// SIMATIC S7-200 project (STEP 7-Micro/WIN), CPU 224XP REL 02.01

SYMBOL_TABLE 输入
一号泵故障            I0.0     // 1号水泵工频故障
二号泵故障            I0.1     // 2号水泵工频故障
三号泵故障            I0.2     // 3号水泵工频故障
一号泵变频运行反馈        I0.3     // 1号水泵变频接触器辅助常开触点
一号泵工频运行反馈        I0.4     // 1号水泵工频接触器辅助常开触点
二号泵变频运行反馈        I0.5     // 2号水泵变频接触器辅助常开触点
二号泵工频运行反馈        I0.6     // 2号水泵工频接触器辅助常开触点
三号泵变频运行反馈        I0.7     // 3号水泵变频接触器辅助常开触点
三号泵工频运行反馈        I1.0     // 3号水泵工频接触器辅助常开触点
变频运行             I1.1     // 变频器准备就绪
变频故障             I1.2     // 变频器故障
自动切换             I1.3     // 变频器达到最大频率
急停               I1.5     // 急停
远方起动             I2.0     // 远方起动系统
水位下限             I2.1     // 水源低水位限位开关
水位上限             I2.2     // 水源高水位限位开关
供水方式             I2.3     // 生活用水/消防用水切换，触点常开为生活用水工作方式
压力测量             AIW0     // 管网压力传感器测量值:4-20mA
END_SYMBOL_TABLE

SYMBOL_TABLE 输出
一号泵变频运行          Q0.0     // 1号水泵变频接触器
一号泵工频运行          Q0.1     // 1号水泵工频接触器
二号泵变频运行          Q0.2     // 2号水泵变频接触器
二号泵工频运行          Q0.3     // 2号水泵工频接触器
三号泵变频运行          Q0.4     // 3号水泵变频接触器
三号泵工频运行          Q0.5     // 3号水泵工频接触器
准备就绪             Q0.6     // 系统准备就绪
报警信号             Q0.7     // 系统报警信号
故障跳闸             Q1.0     // 系统故障跳闸
起动停止             Q1.1     // 变频器起动/停止
供水电磁阀            Q2.0     // 生活用水/消防用水电磁阀控制
频率复位             Q2.1     // 变频器频率复位控制
模拟输出             AQW0     // 变频器模拟输入，PID运算结果: 4-20mA
END_SYMBOL_TABLE

SYMBOL_TABLE PLC內部继电器
允许启动             M1.0     // 系统准备就绪指示
低水位报警            M1.1     // 低水位报警铃声，信号指示
变频报警             M1.2     // 变频器报警铃声，信号指示
火灾报警             M1.3     // 火灾报警铃声，信号指示
HMI急停            M1.5     // 触摸屏急停按钮
远方变频起动自保         M1.6     // 远方变频起动信号自保持
故障结束脉冲           M0.0     // 故障结束脉冲信号
变频起动脉冲           M0.1     // 泵变频启动脉冲
水泵轮换             M0.3     // 倒泵变频启动脉冲
复位变频运行脉冲         M0.4     // 复位当前变频泵运行脉冲
当前泵工频            M0.5     // 当前泵工频运行启动脉冲
新增泵变频            M0.6     // 新泵变频启动脉冲
工变频切换1           M2.0     // 水泵工频/变频转换逻辑控制
工变频切换2           M2.1     // 水泵工频/变频转换逻辑控制
工变频切换3           M2.2     // 水泵工频/变频转换逻辑控制
系统故障             M3.0     // 故障汇总
低水位自保            M3.1     // 低水位自保，高水位复位解除
低水位消铃            M3.2     // 低水位报警铃声消音
变频报警消铃           M3.3     // 变频器故障报警铃声消音
火灾报警消铃           M3.4     // 火灾报警铃声消音
一号泵故障指示          M3.5     // 1号水泵电机过载
二号泵故障指示          M3.6     // 2号水泵电机过载
三号泵故障指示          M3.7     // 3号水泵电机过载
故障复位             M4.1     // 故障自锁信号解除
系统报警指示           M4.2     // 报警汇总
报警确认             M4.3     // 报警自锁信号解除
消铃按钮             M4.4     // 报警铃声信号解除
试灯按钮             M4.5     // 检查报警灯光回路
本地/远方            M5.0     // 触摸屏控制/远方集中控制选择: 默认为本地控制
手动/自动            M5.1     // 工频手动/变频自动: 默认为自动控制
一号泵起动按钮          M5.2     // 触摸屏上1号泵起动按钮
一号泵停止按钮          M6.0     // 触摸屏上1号泵停止按钮
一号泵自保持           M6.1     // 1号泵起动信号自保持
二号泵起动按钮          M6.2     // 触摸屏上2号泵起动按钮
二号泵停止按钮          M6.3     // 触摸屏上2号泵停止按钮
二号泵自保持           M6.4     // 2号泵起动信号自保持
三号泵起动按钮          M6.5     // 触摸屏上3号泵起动按钮
三号泵停止按钮          M6.6     // 触摸屏上3号泵停止按钮
三号泵自保持           M6.7     // 3号泵起动信号自保持
                 M7.0     // 触摸屏变频器起动按钮
                 M7.1     // 触摸屏变频器停止按钮
END_SYMBOL_TABLE

SYMBOL_TABLE PLC內部存储器
压力设置             VW0      // 管网压力设置值
水压测量             VW2      // 管网压力传感器测量值
过程变量             VD100
压力给定             VD104
PI计算值            VD108
比例系数             VD112
采样时间             VD116
积分时间             VD120
微分时间             VD124
频率下限             VD204    // 变频运行频率下限值
生活水频率上限          VD208    // 生活供水变频运行频率上限值
消防水频率上限          VD212    // 消防供水变频运行频率上限值
PI调节值            VD250    // PI调节结果存储器
变频泵号             VD300    // 记录当前变频工作泵的泵号
工频泵总数            VD301    // 工频运行泵的总数量
泵轮换时间            VD310    // 变频泵运行时间存储器
工频变频切换1          T33      // 水泵工频/变频转换逻辑时间控制
工频变频切换2          T34      // 水泵工频/变频转换逻辑时间控制
工频变频切换3          T39      // 水泵工频/变频转换逻辑时间控制
工频增泵时间           T37      // 工频泵增泵滤波时间控制
工频减泵时间           T38      // 工频泵减泵滤波时间控制
END_SYMBOL_TABLE

SYMBOL_TABLE S7-200 符号
Always_On        SM0.0    // 始终接通为 ON
First_Scan_On    SM0.1    // 仅第一个扫描周期中接通为 ON
Clock_60s        SM0.4    // 在 1 分钟的循环周期内，接通为 ON 30  秒，关断为 OFF 30 秒
Clock_1s         SM0.5    // 在 1 秒钟的循环周期内，接通为 ON 0.5 秒，关断为 OFF 0.5  秒
Time_0_Intrvl    SMB34    // 定时中断 0 的时间间隔（从 1 至 255，以 1 毫秒为增量）。
END_SYMBOL_TABLE

ORGANIZATION_BLOCK 主程序:OB1
TITLE=程序注释
BEGIN
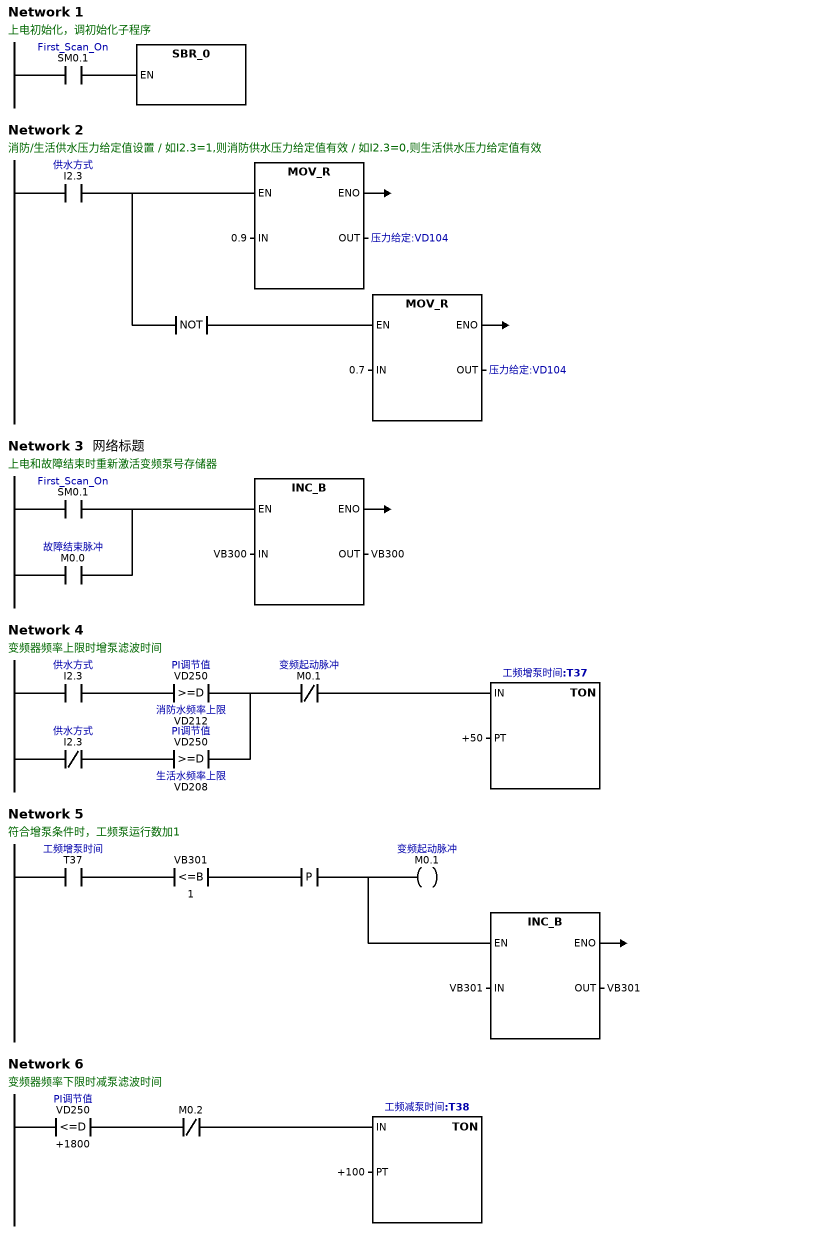
Network 1
// 上电初始化，调初始化子程序
// (network saved uncompiled; LAD cells follow)
// row 0: c0 -| |- First_Scan_On:SM0.1  c1 [SBR_0 EN:=power@row0]
Network 2
// 消防/生活供水压力给定值设置
// 如I2.3=1,则消防供水压力给定值有效
// 如I2.3=0,则生活供水压力给定值有效
// (network saved uncompiled; LAD cells follow)
// row 0: c0 -| |- 供水方式:I2.3 v  c1 --  c2 [MOV_R EN:=power@row0, IN:=0.9, ENO=>power, OUT=>压力给定:VD104]  c3 ->
// row 1: c0 ^v  c2 [box]
// row 2: c0 ^  c1 -|NOT|-  c2 --  c3 [MOV_R EN:=power@row2, IN:=0.7, ENO=>power, OUT=>压力给定:VD104]  c4 ->
// row 3: c3 [box]
Network 3 // 网络标题
// 上电和故障结束时重新激活变频泵号存储器
// (network saved uncompiled; LAD cells follow)
// row 0: c0 -| |- First_Scan_On:SM0.1 v  c1 --  c2 [INC_B EN:=power@row0, IN:=VB300, ENO=>power, OUT=>VB300]  c3 ->
// row 1: c0 -| |- 故障结束脉冲:M0.0 ^  c2 [box]
Network 4
// 变频器频率上限时增泵滤波时间
// (network saved uncompiled; LAD cells follow)
// row 0: c0 -| |- 供水方式:I2.3  c1 -|>=D|- PI调节值:VD250, 消防水频率上限:VD212 v  c2 -|/|- 变频起动脉冲:M0.1  c3 --  c4 [TON 工频增泵时间:T37 IN:=power@row0, PT:=+50]
// row 1: c0 -|/|- 供水方式:I2.3  c1 -|>=D|- PI调节值:VD250, 生活水频率上限:VD208 ^  c4 [box]
Network 5
// 符合增泵条件时，工频泵运行数加1
// (network saved uncompiled; LAD cells follow)
// row 0: c0 -| |- 工频增泵时间:T37  c1 -|<=B|- VB301, 1  c2 -|P|-  v  c3 -( ) 变频起动脉冲:M0.1
// row 1: c2 ^  c3 --  c4 [INC_B EN:=power@row1, IN:=VB301, ENO=>power, OUT=>VB301]  c5 ->
// row 2: c4 [box]
Network 6
// 变频器频率下限时减泵滤波时间
// (network saved uncompiled; LAD cells follow)
// row 0: c0 -|<=D|- PI调节值:VD250, +1800  c1 -|/|- M0.2  c2 --  c3 [TON 工频减泵时间:T38 IN:=power@row0, PT:=+100]
// row 1: c3 [box]
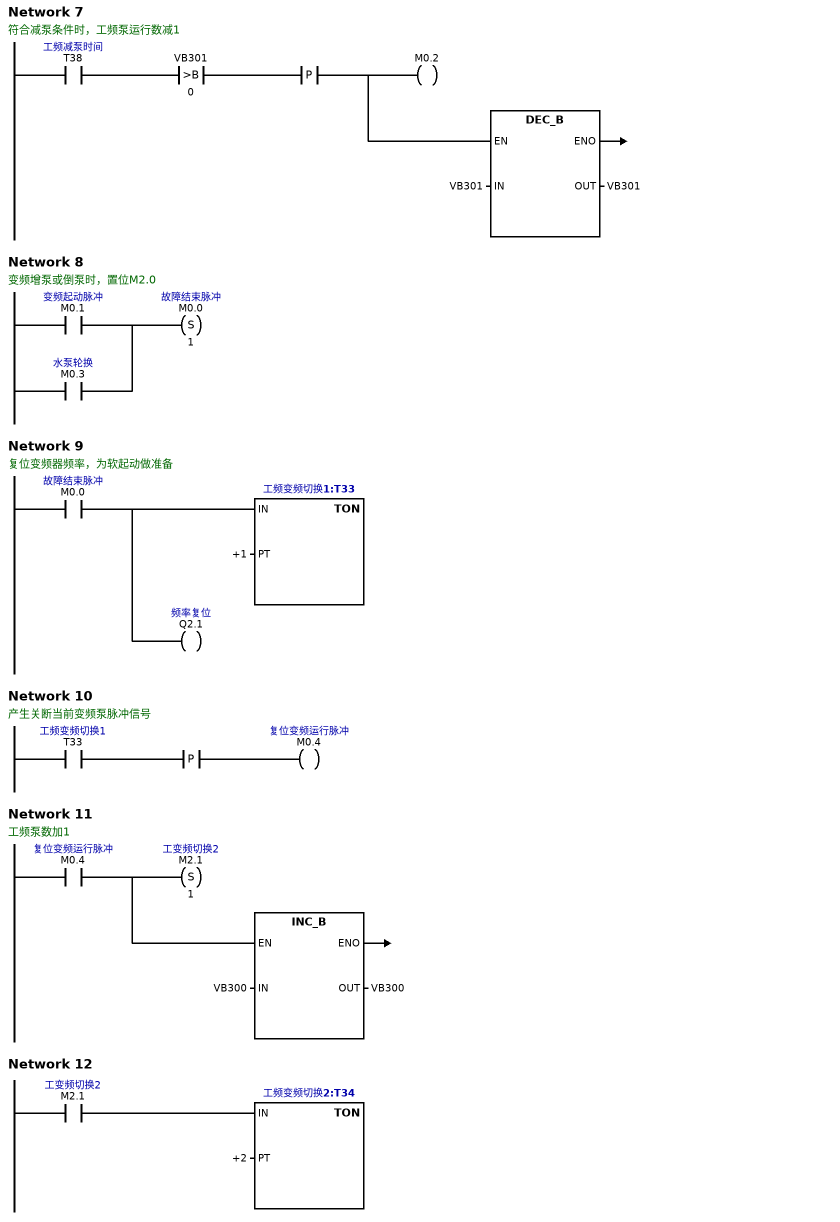
Network 7
// 符合减泵条件时，工频泵运行数减1
// (network saved uncompiled; LAD cells follow)
// row 0: c0 -| |- 工频减泵时间:T38  c1 -|>B|- VB301, 0  c2 -|P|-  v  c3 -( ) M0.2
// row 1: c2 ^  c3 --  c4 [DEC_B EN:=power@row1, IN:=VB301, ENO=>power, OUT=>VB301]  c5 ->
// row 2: c4 [box]
Network 8
// 变频增泵或倒泵时，置位M2.0
// (network saved uncompiled; LAD cells follow)
// row 0: c0 -| |- 变频起动脉冲:M0.1 v  c1 -(S) 故障结束脉冲:M0.0, 1
// row 1: c0 -| |- 水泵轮换:M0.3 ^
Network 9
// 复位变频器频率，为软起动做准备
// (network saved uncompiled; LAD cells follow)
// row 0: c0 -| |- 故障结束脉冲:M0.0 v  c1 --  c2 [TON 工频变频切换1:T33 IN:=power@row0, PT:=+1]
// row 1: c0 ^v  c2 [box]
// row 2: c0 ^  c1 -( ) 频率复位:Q2.1
Network 10
// 产生关断当前变频泵脉冲信号
// (network saved uncompiled; LAD cells follow)
// row 0: c0 -| |- 工频变频切换1:T33  c1 -|P|-  c2 -( ) 复位变频运行脉冲:M0.4
Network 11
// 工频泵数加1
// (network saved uncompiled; LAD cells follow)
// row 0: c0 -| |- 复位变频运行脉冲:M0.4 v  c1 -(S) 工变频切换2:M2.1, 1
// row 1: c0 ^  c1 --  c2 [INC_B EN:=power@row1, IN:=VB300, ENO=>power, OUT=>VB300]  c3 ->
// row 2: c2 [box]
Network 12
// (network saved uncompiled; LAD cells follow)
// row 0: c0 -| |- 工变频切换2:M2.1  c1 --  c2 [TON 工频变频切换2:T34 IN:=power@row0, PT:=+2]
// row 1: c2 [box]
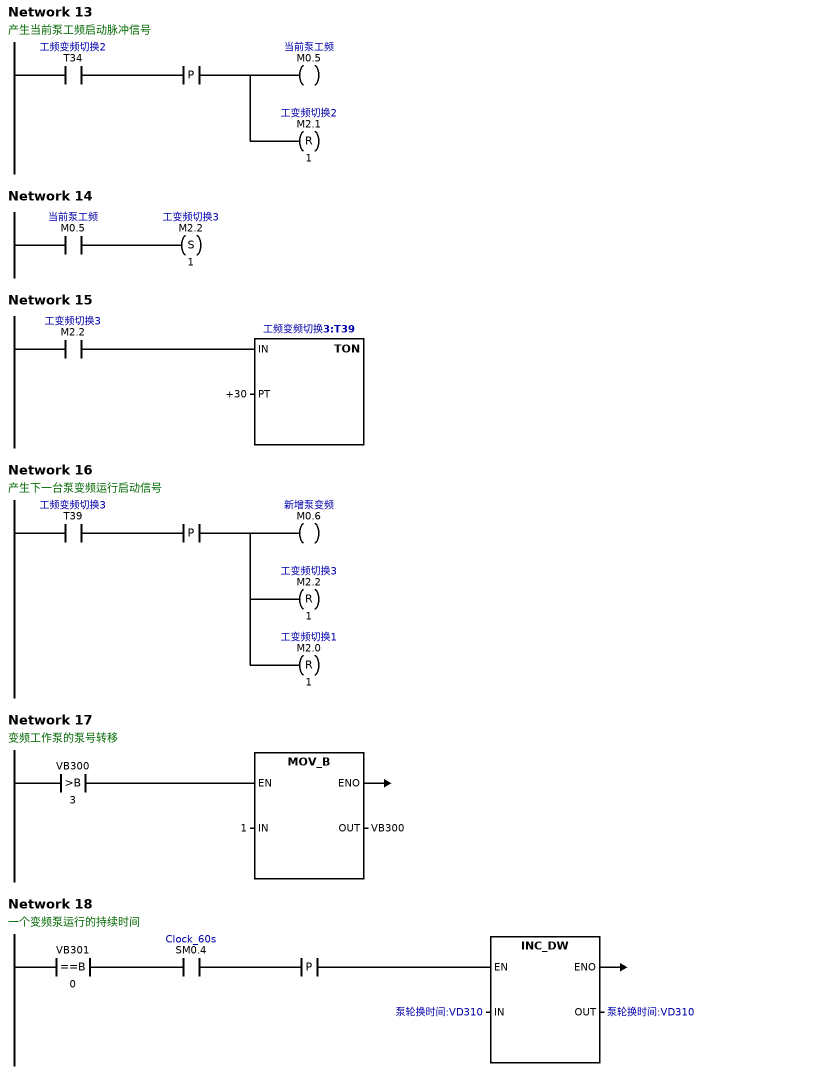
Network 13
// 产生当前泵工频启动脉冲信号
// (network saved uncompiled; LAD cells follow)
// row 0: c0 -| |- 工频变频切换2:T34  c1 -|P|-  v  c2 -( ) 当前泵工频:M0.5
// row 1: c1 ^  c2 -(R) 工变频切换2:M2.1, 1
Network 14
// (network saved uncompiled; LAD cells follow)
// row 0: c0 -| |- 当前泵工频:M0.5  c1 -(S) 工变频切换3:M2.2, 1
Network 15
// (network saved uncompiled; LAD cells follow)
// row 0: c0 -| |- 工变频切换3:M2.2  c1 --  c2 [TON 工频变频切换3:T39 IN:=power@row0, PT:=+30]
// row 1: c2 [box]
Network 16
// 产生下一台泵变频运行启动信号
// (network saved uncompiled; LAD cells follow)
// row 0: c0 -| |- 工频变频切换3:T39  c1 -|P|-  v  c2 -( ) 新增泵变频:M0.6
// row 1: c1 ^v  c2 -(R) 工变频切换3:M2.2, 1
// row 2: c1 ^  c2 -(R) 工变频切换1:M2.0, 1
Network 17
// 变频工作泵的泵号转移
LDB>   VB300, 3
MOVB   1, VB300
Network 18
// 一个变频泵运行的持续时间
LDB=   VB301, 0
A      Clock_60s:SM0.4
EU
INCD   泵轮换时间:VD310
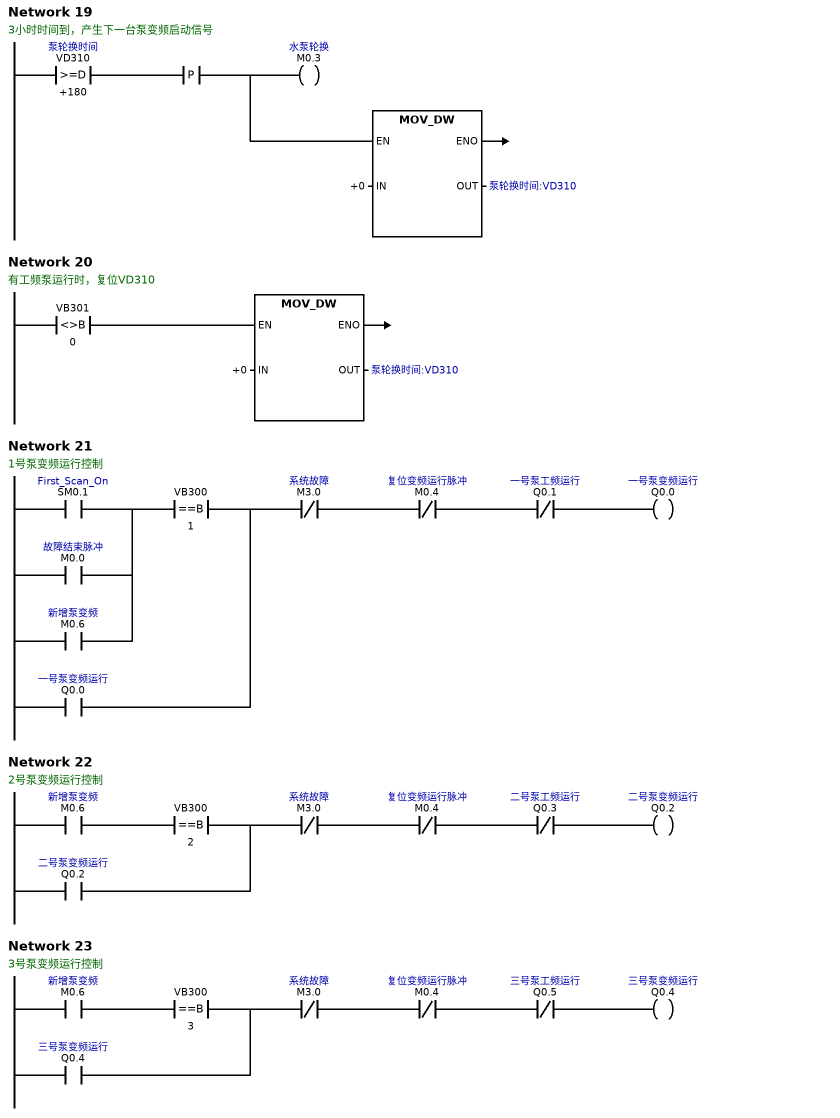
Network 19
// 3小时时间到，产生下一台泵变频启动信号
// (network saved uncompiled; LAD cells follow)
// row 0: c0 -|>=D|- 泵轮换时间:VD310, +180  c1 -|P|-  v  c2 -( ) 水泵轮换:M0.3
// row 1: c1 ^  c2 --  c3 [MOV_DW EN:=power@row1, IN:=+0, ENO=>power, OUT=>泵轮换时间:VD310]  c4 ->
// row 2: c3 [box]
Network 20
// 有工频泵运行时，复位VD310
LDB<>  VB301, 0
MOVD   +0, 泵轮换时间:VD310
Network 21
// 1号泵变频运行控制
// (network saved uncompiled; LAD cells follow)
// row 0: c0 -| |- First_Scan_On:SM0.1 v  c1 -|==B|- VB300, 1 v  c2 -|/|- 系统故障:M3.0  c3 -|/|- 复位变频运行脉冲:M0.4  c4 -|/|- 一号泵工频运行:Q0.1  c5 -( ) 一号泵变频运行:Q0.0
// row 1: c0 -| |- 故障结束脉冲:M0.0 ^v  c1 ^v
// row 2: c0 -| |- 新增泵变频:M0.6 ^  c1 ^v
// row 3: c0 -| |- 一号泵变频运行:Q0.0  c1 -- ^
Network 22
// 2号泵变频运行控制
// (network saved uncompiled; LAD cells follow)
// row 0: c0 -| |- 新增泵变频:M0.6  c1 -|==B|- VB300, 2 v  c2 -|/|- 系统故障:M3.0  c3 -|/|- 复位变频运行脉冲:M0.4  c4 -|/|- 二号泵工频运行:Q0.3  c5 -( ) 二号泵变频运行:Q0.2
// row 1: c0 -| |- 二号泵变频运行:Q0.2  c1 -- ^
Network 23
// 3号泵变频运行控制
// (network saved uncompiled; LAD cells follow)
// row 0: c0 -| |- 新增泵变频:M0.6  c1 -|==B|- VB300, 3 v  c2 -|/|- 系统故障:M3.0  c3 -|/|- 复位变频运行脉冲:M0.4  c4 -|/|- 三号泵工频运行:Q0.5  c5 -( ) 三号泵变频运行:Q0.4
// row 1: c0 -| |- 三号泵变频运行:Q0.4  c1 -- ^
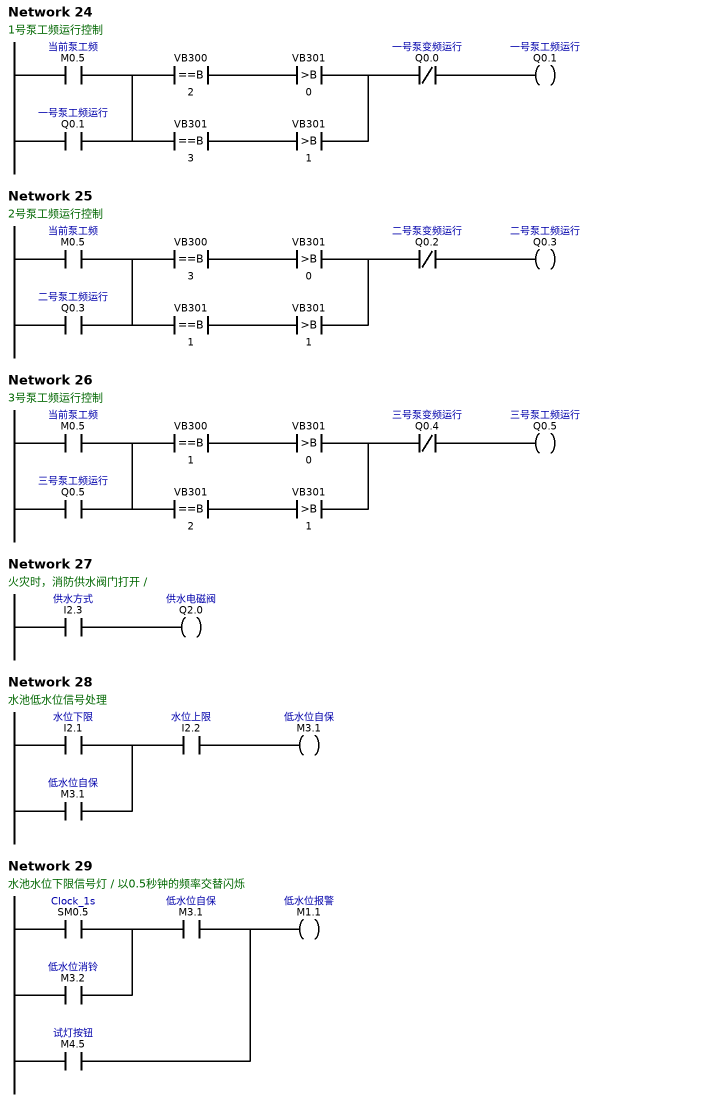
Network 24
// 1号泵工频运行控制
// (network saved uncompiled; LAD cells follow)
// row 0: c0 -| |- 当前泵工频:M0.5 v  c1 -|==B|- VB300, 2  c2 -|>B|- VB301, 0 v  c3 -|/|- 一号泵变频运行:Q0.0  c4 -( ) 一号泵工频运行:Q0.1
// row 1: c0 -| |- 一号泵工频运行:Q0.1 ^  c1 -|==B|- VB301, 3  c2 -|>B|- VB301, 1 ^
Network 25
// 2号泵工频运行控制
// (network saved uncompiled; LAD cells follow)
// row 0: c0 -| |- 当前泵工频:M0.5 v  c1 -|==B|- VB300, 3  c2 -|>B|- VB301, 0 v  c3 -|/|- 二号泵变频运行:Q0.2  c4 -( ) 二号泵工频运行:Q0.3
// row 1: c0 -| |- 二号泵工频运行:Q0.3 ^  c1 -|==B|- VB301, 1  c2 -|>B|- VB301, 1 ^
Network 26
// 3号泵工频运行控制
// (network saved uncompiled; LAD cells follow)
// row 0: c0 -| |- 当前泵工频:M0.5 v  c1 -|==B|- VB300, 1  c2 -|>B|- VB301, 0 v  c3 -|/|- 三号泵变频运行:Q0.4  c4 -( ) 三号泵工频运行:Q0.5
// row 1: c0 -| |- 三号泵工频运行:Q0.5 ^  c1 -|==B|- VB301, 2  c2 -|>B|- VB301, 1 ^
Network 27
// 火灾时，消防供水阀门打开
// 
// (network saved uncompiled; LAD cells follow)
// row 0: c0 -| |- 供水方式:I2.3  c1 -( ) 供水电磁阀:Q2.0
Network 28
// 水池低水位信号处理
// (network saved uncompiled; LAD cells follow)
// row 0: c0 -| |- 水位下限:I2.1 v  c1 -| |- 水位上限:I2.2  c2 -( ) 低水位自保:M3.1
// row 1: c0 -| |- 低水位自保:M3.1 ^
Network 29
// 水池水位下限信号灯
// 以0.5秒钟的频率交替闪烁
// (network saved uncompiled; LAD cells follow)
// row 0: c0 -| |- Clock_1s:SM0.5 v  c1 -| |- 低水位自保:M3.1 v  c2 -( ) 低水位报警:M1.1
// row 1: c0 -| |- 低水位消铃:M3.2 ^  c1 ^v
// row 2: c0 -| |- 试灯按钮:M4.5  c1 -- ^
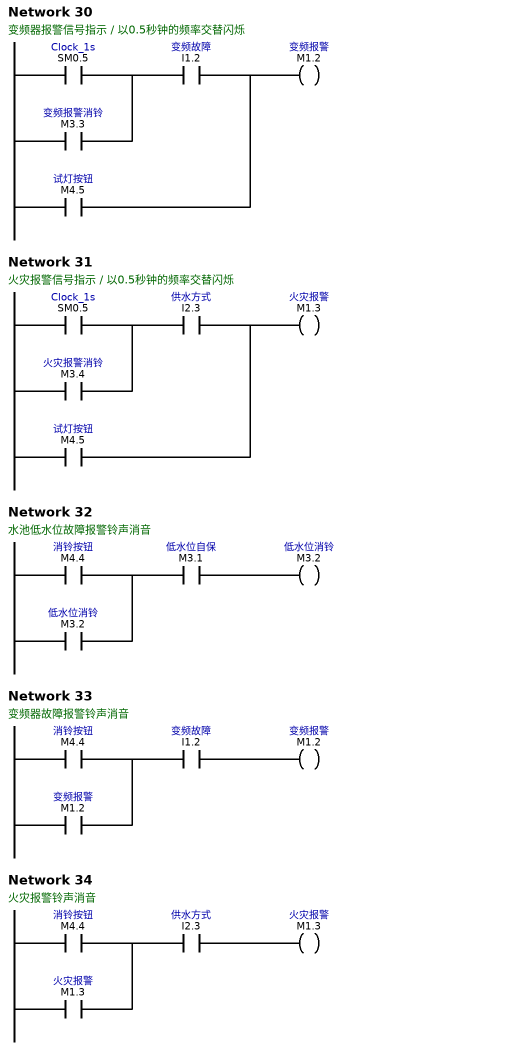
Network 30
// 变频器报警信号指示
// 以0.5秒钟的频率交替闪烁
// (network saved uncompiled; LAD cells follow)
// row 0: c0 -| |- Clock_1s:SM0.5 v  c1 -| |- 变频故障:I1.2 v  c2 -( ) 变频报警:M1.2
// row 1: c0 -| |- 变频报警消铃:M3.3 ^  c1 ^v
// row 2: c0 -| |- 试灯按钮:M4.5  c1 -- ^
Network 31
// 火灾报警信号指示
// 以0.5秒钟的频率交替闪烁
// (network saved uncompiled; LAD cells follow)
// row 0: c0 -| |- Clock_1s:SM0.5 v  c1 -| |- 供水方式:I2.3 v  c2 -( ) 火灾报警:M1.3
// row 1: c0 -| |- 火灾报警消铃:M3.4 ^  c1 ^v
// row 2: c0 -| |- 试灯按钮:M4.5  c1 -- ^
Network 32
// 水池低水位故障报警铃声消音
// (network saved uncompiled; LAD cells follow)
// row 0: c0 -| |- 消铃按钮:M4.4 v  c1 -| |- 低水位自保:M3.1  c2 -( ) 低水位消铃:M3.2
// row 1: c0 -| |- 低水位消铃:M3.2 ^
Network 33
// 变频器故障报警铃声消音
// (network saved uncompiled; LAD cells follow)
// row 0: c0 -| |- 消铃按钮:M4.4 v  c1 -| |- 变频故障:I1.2  c2 -( ) 变频报警:M1.2
// row 1: c0 -| |- 变频报警:M1.2 ^
Network 34
// 火灾报警铃声消音
// (network saved uncompiled; LAD cells follow)
// row 0: c0 -| |- 消铃按钮:M4.4 v  c1 -| |- 供水方式:I2.3  c2 -( ) 火灾报警:M1.3
// row 1: c0 -| |- 火灾报警:M1.3 ^
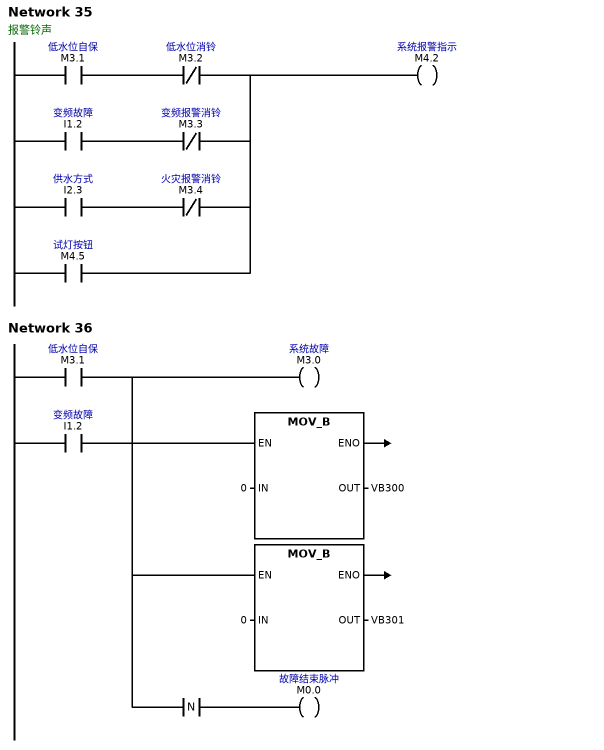
Network 35
// 报警铃声
// (network saved uncompiled; LAD cells follow)
// row 0: c0 -| |- 低水位自保:M3.1  c1 -|/|- 低水位消铃:M3.2 v  c2 --  c3 -( ) 系统报警指示:M4.2
// row 1: c0 -| |- 变频故障:I1.2  c1 -|/|- 变频报警消铃:M3.3 ^v
// row 2: c0 -| |- 供水方式:I2.3  c1 -|/|- 火灾报警消铃:M3.4 ^v
// row 3: c0 -| |- 试灯按钮:M4.5  c1 -- ^
Network 36
// (network saved uncompiled; LAD cells follow)
// row 0: c0 -| |- 低水位自保:M3.1 v  c1 --  c2 -( ) 系统故障:M3.0
// row 1: c0 -| |- 变频故障:I1.2 ^v  c1 --  c2 [MOV_B EN:=power@row1, IN:=0, ENO=>power, OUT=>VB300]  c3 ->
// row 2: c0 ^v  c2 [box]
// row 3: c0 ^v  c1 --  c2 [MOV_B EN:=power@row3, IN:=0, ENO=>power, OUT=>VB301]  c3 ->
// row 4: c0 ^v  c2 [box]
// row 5: c0 ^  c1 -|N|-  c2 -( ) 故障结束脉冲:M0.0
Network 37 // 网络标题
Network 38 // 网络标题
// 网络注释
END_ORGANIZATION_BLOCK

SUBROUTINE_BLOCK SBR_0:SBR0
TITLE=子程序注释
BEGIN
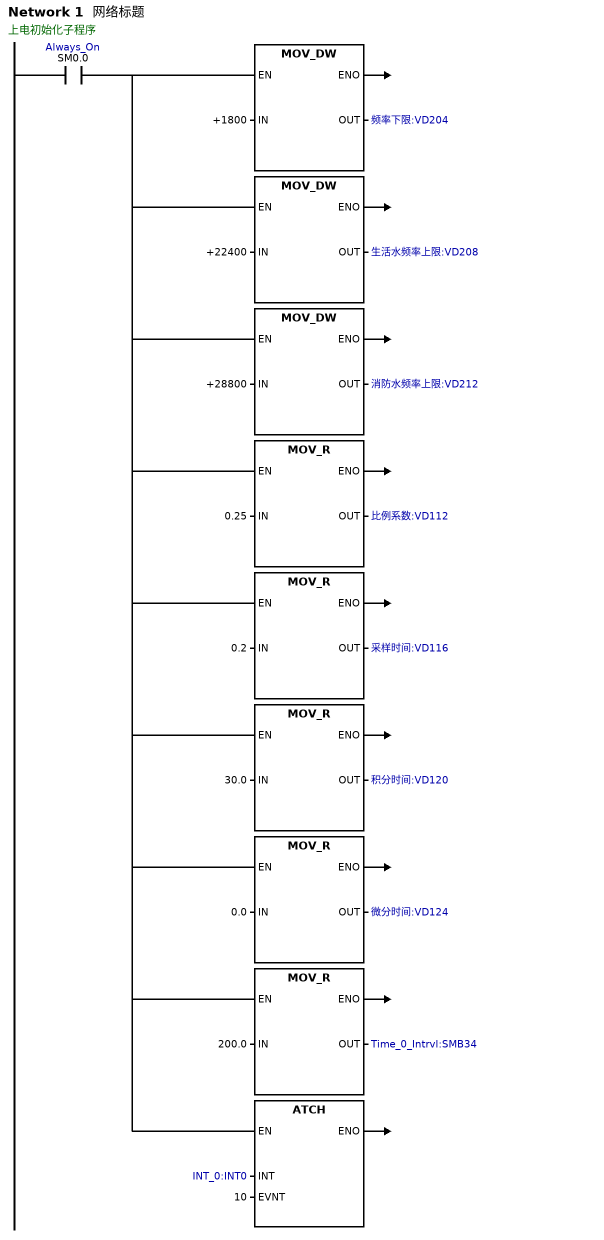
Network 1 // 网络标题
// 上电初始化子程序
// (network saved uncompiled; LAD cells follow)
// row 0: c0 -| |- Always_On:SM0.0 v  c1 --  c2 [MOV_DW EN:=power@row0, IN:=+1800, ENO=>power, OUT=>频率下限:VD204]  c3 ->
// row 1: c0 ^v  c2 [box]
// row 2: c0 ^v  c1 --  c2 [MOV_DW EN:=power@row2, IN:=+22400, ENO=>power, OUT=>生活水频率上限:VD208]  c3 ->
// row 3: c0 ^v  c2 [box]
// row 4: c0 ^v  c1 --  c2 [MOV_DW EN:=power@row4, IN:=+28800, ENO=>power, OUT=>消防水频率上限:VD212]  c3 ->
// row 5: c0 ^v  c2 [box]
// row 6: c0 ^v  c1 --  c2 [MOV_R EN:=power@row6, IN:=0.25, ENO=>power, OUT=>比例系数:VD112]  c3 ->
// row 7: c0 ^v  c2 [box]
// row 8: c0 ^v  c1 --  c2 [MOV_R EN:=power@row8, IN:=0.2, ENO=>power, OUT=>采样时间:VD116]  c3 ->
// row 9: c0 ^v  c2 [box]
// row 10: c0 ^v  c1 --  c2 [MOV_R EN:=power@row10, IN:=30.0, ENO=>power, OUT=>积分时间:VD120]  c3 ->
// row 11: c0 ^v  c2 [box]
// row 12: c0 ^v  c1 --  c2 [MOV_R EN:=power@row12, IN:=0.0, ENO=>power, OUT=>微分时间:VD124]  c3 ->
// row 13: c0 ^v  c2 [box]
// row 14: c0 ^v  c1 --  c2 [MOV_R EN:=power@row14, IN:=200.0, ENO=>power, OUT=>Time_0_Intrvl:SMB34]  c3 ->
// row 15: c0 ^v  c2 [box]
// row 16: c0 ^  c1 --  c2 [ATCH EN:=power@row16, INT:=INT_0:INT0, EVNT:=10, ENO=>power]  c3 ->
// row 17: c2 [box]
END_SUBROUTINE_BLOCK

INTERRUPT_BLOCK INT_0:INT0
TITLE=中断程序注释
BEGIN
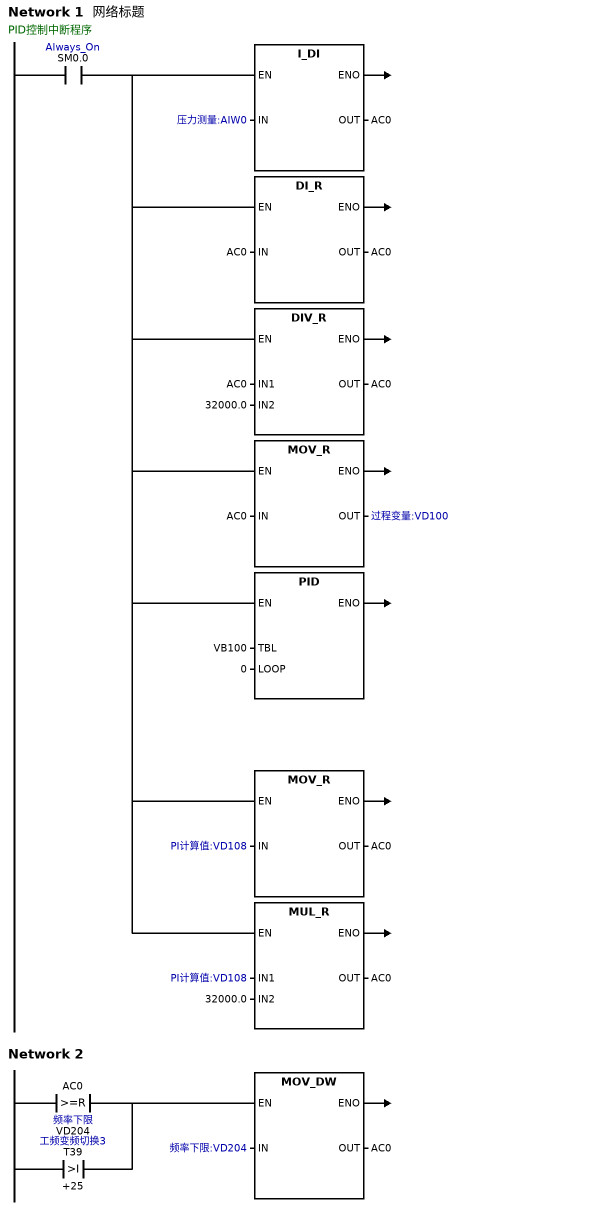
Network 1 // 网络标题
// PID控制中断程序
// (network saved uncompiled; LAD cells follow)
// row 0: c0 -| |- Always_On:SM0.0 v  c1 --  c2 [I_DI EN:=power@row0, IN:=压力测量:AIW0, ENO=>power, OUT=>AC0]  c3 ->
// row 1: c0 ^v  c2 [box]
// row 2: c0 ^v  c1 --  c2 [DI_R EN:=power@row2, IN:=AC0, ENO=>power, OUT=>AC0]  c3 ->
// row 3: c0 ^v  c2 [box]
// row 4: c0 ^v  c1 --  c2 [DIV_R EN:=power@row4, IN1:=AC0, IN2:=32000.0, ENO=>power, OUT=>AC0]  c3 ->
// row 5: c0 ^v  c2 [box]
// row 6: c0 ^v  c1 --  c2 [MOV_R EN:=power@row6, IN:=AC0, ENO=>power, OUT=>过程变量:VD100]  c3 ->
// row 7: c0 ^v  c2 [box]
// row 8: c0 ^v  c1 --  c2 [PID EN:=power@row8, TBL:=VB100, LOOP:=0, ENO=>power]  c3 ->
// row 9: c0 ^v  c2 [box]
// row 10: c0 ^v
// row 11: c0 ^v  c1 --  c2 [MOV_R EN:=power@row11, IN:=PI计算值:VD108, ENO=>power, OUT=>AC0]  c3 ->
// row 12: c0 ^v  c2 [box]
// row 13: c0 ^  c1 --  c2 [MUL_R EN:=power@row13, IN1:=PI计算值:VD108, IN2:=32000.0, ENO=>power, OUT=>AC0]  c3 ->
// row 14: c2 [box]
Network 2
// (network saved uncompiled; LAD cells follow)
// row 0: c0 -|>=R|- AC0, 频率下限:VD204 v  c1 --  c2 [MOV_DW EN:=power@row0, IN:=频率下限:VD204, ENO=>power, OUT=>AC0]  c3 ->
// row 1: c0 -|>I|- 工频变频切换3:T39, +25 ^  c2 [box]
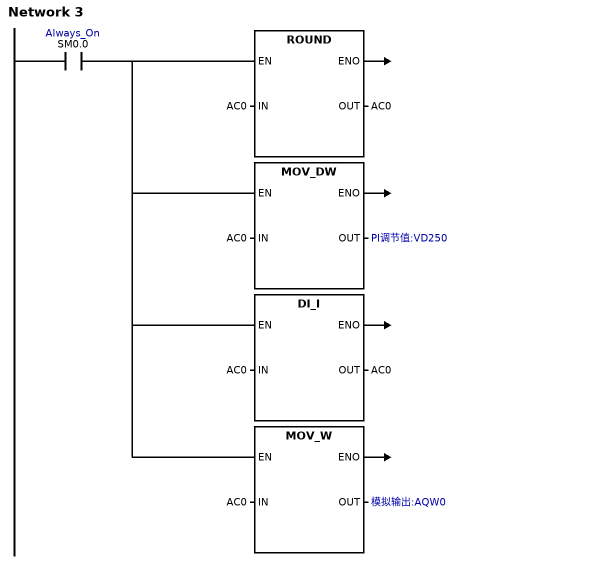
Network 3
// (network saved uncompiled; LAD cells follow)
// row 0: c0 -| |- Always_On:SM0.0 v  c1 --  c2 [ROUND EN:=power@row0, IN:=AC0, ENO=>power, OUT=>AC0]  c3 ->
// row 1: c0 ^v  c2 [box]
// row 2: c0 ^v  c1 --  c2 [MOV_DW EN:=power@row2, IN:=AC0, ENO=>power, OUT=>PI调节值:VD250]  c3 ->
// row 3: c0 ^v  c2 [box]
// row 4: c0 ^v  c1 --  c2 [DI_I EN:=power@row4, IN:=AC0, ENO=>power, OUT=>AC0]  c3 ->
// row 5: c0 ^v  c2 [box]
// row 6: c0 ^  c1 --  c2 [MOV_W EN:=power@row6, IN:=AC0, ENO=>power, OUT=>模拟输出:AQW0]  c3 ->
// row 7: c2 [box]
END_INTERRUPT_BLOCK
